(* IEC 61131-3 sources: s22-soft-shell/st_interpret/tests/test_inputs/execution/st_subset_3-4, 5 files *)

(* ---- 03_add.st ---- *)
PROGRAM 03_Add
VAR
    a: int;
    ST_TESTING_RESULT : bool;
END_VAR
a := (1 + 2);
        ST_TESTING_RESULT := (a = 3);
END_PROGRAM

(* ---- 03_sub.st ---- *)
PROGRAM 03_Sub
VAR
    a: int;
    ST_TESTING_RESULT : bool;
END_VAR
a := (2 - 1);
        ST_TESTING_RESULT := (a = 1);
END_PROGRAM

(* ---- 04_div.st ---- *)
PROGRAM 04_div
VAR
    a: int;
    ST_TESTING_RESULT : bool;
END_VAR
a := (10 / 2);
        ST_TESTING_RESULT := (a = 5);
END_PROGRAM

(* ---- 04_mul.st ---- *)
PROGRAM 04_mul
VAR
    a: int;
    ST_TESTING_RESULT : bool;
END_VAR
a := (3 * 2);
        ST_TESTING_RESULT := (a = 6);
END_PROGRAM

(* ---- 04_testA.st ---- *)
PROGRAM 04_testA
VAR
    a: int;
    ST_TESTING_RESULT : bool;
END_VAR
a := (2 + 4) * (1 + 3);
        ST_TESTING_RESULT := (a = 24);
END_PROGRAM
